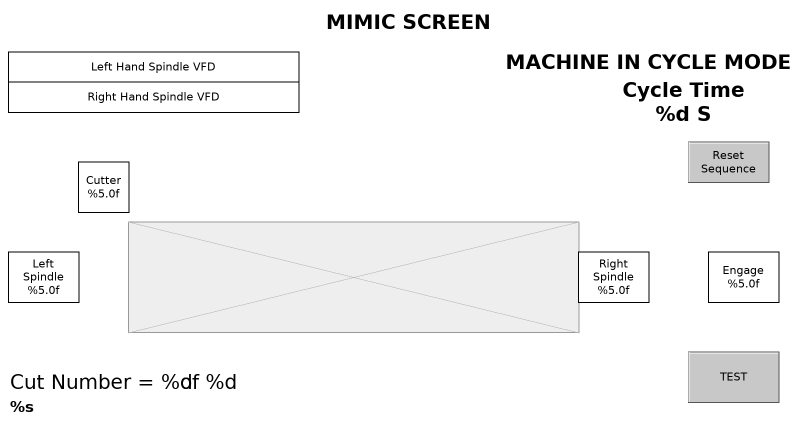
bitmap at (130,220)-(581,331): c:\users\graemep\pictures\bellow.bmp
rectangle at (80,160)-(131,211): text "Cutter / %5.0f"; shows MAIN.Axis[4].nActualPosition; x offset HMI.nCutterSlideXOffset; y offset HMI.nCutterYOffset; scale 1000
rectangle at (710,250)-(781,301): text "Engage / %5.0f"; shows MAIN.Axis[5].nActualPosition; x offset -HMI.nEnagageXOffset; y offset 0; scale 1000
rectangle at (580,250)-(651,301): text "Right / Spindle / %5.0f"; shows MAIN.Axis[2].nActualPosition; alarm colour if MAIN.bAxis2Coupled; x offset HMI.nRightSpindleXOffset; y offset 0; scale 1000
rectangle at (10,360)-(191,401): text "Cut Number = %d"; shows Sequencer.nCurrentCutNumber; invisible if .nMachineType = SIZER
button at (690,350)-(781,401): text "TEST"; invisible if .CurrentUserLevel < 2; taps Sequencer.bHMI_Overide
rectangle at (10,390)-(511,421): text "%s"; shows Sequencer.sSequence_Text
rounded rectangle at (10,50)-(301,81): text "Left Hand Spindle VFD"; invisible if .nMachineType = SIZER; alarm colour if .qbLeftHandSpindleOn
rounded rectangle at (10,80)-(301,111): text "Right Hand Spindle VFD"; invisible if .nMachineType = SIZER; alarm colour if .qbRightHandSpindleOn
rectangle at (10,250)-(81,301): text "Left / Spindle / %5.0f"; shows MAIN.Axis[1].nActualPosition; alarm colour if MAIN.bAxis2Coupled; x offset HMI.nLeftSpindleXOffset; y offset 0; scale 1000
rectangle at (500,40)-(801,81): text "MACHINE IN CYCLE MODE"; invisible if NOT MAIN.bInCycle
rectangle at (620,60)-(751,141): text "Cycle Time / %d S"; shows MAIN.nCycleTime
rectangle at (180,360)-(251,401): text "of %d"; shows .MachineRecipes[nCurrentRecipe].nNumberOfCuts; invisible if .nMachineType = SIZER
rectangle at (320,0)-(501,41): text "MIMIC SCREEN"
button at (690,140)-(771,181): text "Reset / Sequence"; runs INTERN ASSIGN Sequencer.nMachineSequence:=(0)
*)

(* Visualisation Helpers/Motion Helpers/MOVE_TABLE
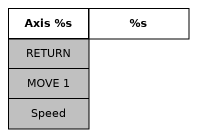
rounded rectangle at (0,30)-(81,61): text "RETURN"
rounded rectangle at (0,60)-(81,91): text "MOVE 1"
rounded rectangle at (0,0)-(81,31): text "Axis %s"; shows $AXISNUMBER$
rounded rectangle at (0,90)-(81,121): text "Speed"
rounded rectangle at (80,0)-(181,31): text "%s"; shows $AXISNAME$
3 elements of other kinds (tables, trends, ...) not read
*)

(* Visualisation Helpers/Motion Helpers/MUILTI_MOVE_TABLE
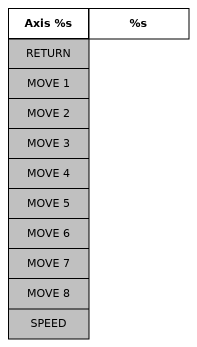
rounded rectangle at (0,30)-(81,61): text "RETURN"
rounded rectangle at (0,60)-(81,91): text "MOVE 1"
rounded rectangle at (0,90)-(81,121): text "MOVE 2"
rounded rectangle at (0,120)-(81,151): text "MOVE 3"
rounded rectangle at (0,150)-(81,181): text "MOVE 4"
rounded rectangle at (0,0)-(81,31): text "Axis %s"; shows $AXISNUMBER$
rounded rectangle at (0,300)-(81,331): text "SPEED"
rounded rectangle at (0,180)-(81,211): text "MOVE 5"
rounded rectangle at (0,210)-(81,241): text "MOVE 6"
rounded rectangle at (0,240)-(81,271): text "MOVE 7"
rounded rectangle at (0,270)-(81,301): text "MOVE 8"
rounded rectangle at (80,0)-(181,31): text "%s"; shows $AXISNAME$
10 elements of other kinds (tables, trends, ...) not read
*)

(* Visualisation Helpers/NUM_PAD
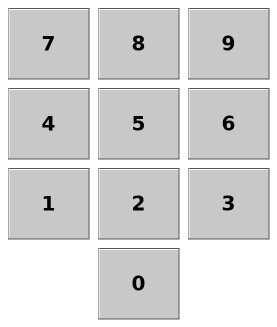
button at (20,20)-(101,91): text "7"; runs INTERN ASSIGN $KEY_PRESSED$:=(7)
button at (110,20)-(191,91): text "8"; runs INTERN ASSIGN $KEY_PRESSED$:=(8)
button at (110,260)-(191,331): text "0"; runs INTERN ASSIGN $KEY_PRESSED$:=(0)
button at (200,20)-(281,91): text "9"; runs INTERN ASSIGN $KEY_PRESSED$:=(9)
button at (20,100)-(101,171): text "4"; runs INTERN ASSIGN $KEY_PRESSED$:=(4)
button at (110,100)-(191,171): text "5"; runs INTERN ASSIGN $KEY_PRESSED$:=(5)
button at (200,100)-(281,171): text "6"; runs INTERN ASSIGN $KEY_PRESSED$:=(6)
button at (20,180)-(101,251): text "1"
button at (110,180)-(191,251): text "2"; runs INTERN ASSIGN $KEY_PRESSED$:=(2)
button at (200,180)-(281,251): text "3"; runs INTERN ASSIGN $KEY_PRESSED$:=(3)
*)

(* Visualisation Helpers/POPUP
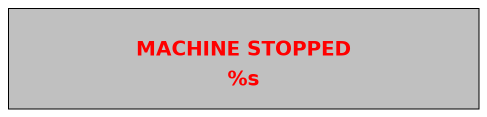
rectangle at (110,20)-(361,61): text "MACHINE STOPPED"; invisible if MAIN.bMachineRunning
rectangle at (20,50)-(451,91): text "%s"; shows Machine.ErrorHandler.sFirstError
2 more shapes without text or variables
*)

(* Visualisation RECIPE_EDITOR
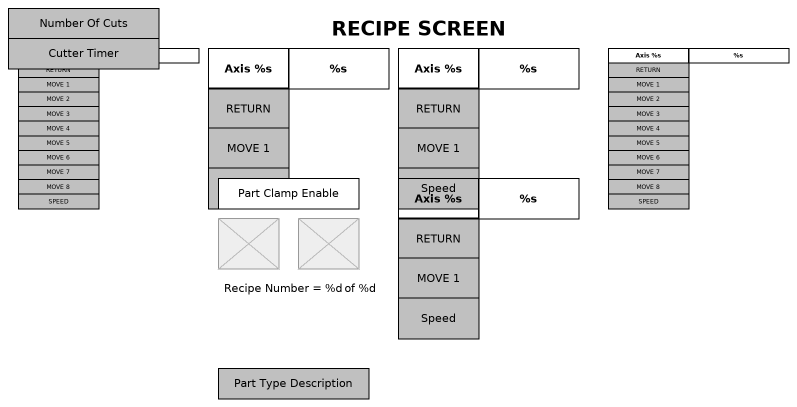
rectangle at (320,0)-(501,41): text "RECIPE SCREEN"
embedded screen at (10,40)-(191,201): MUILTI_MOVE_TABLE
embedded screen at (200,40)-(381,201): MOVE_TABLE
embedded screen at (390,40)-(571,201): MOVE_TABLE
bitmap at (210,210)-(271,261): c:\users\graemep\pictures\imagesi6yb17pr.jpg
bitmap at (290,210)-(351,261): c:\users\graemep\pictures\right arrow.jpg
rectangle at (200,260)-(351,301): text "Recipe Number = %d"; shows nRecipeNumber
embedded screen at (600,40)-(781,201): MUILTI_MOVE_TABLE
embedded screen at (390,170)-(571,331): MOVE_TABLE
rounded rectangle at (210,170)-(351,201): text "Part Clamp Enable"; invisible if .nMachineType = CUTTER; alarm colour if MachineRecipes[nRecipeNumber].bPartClampEnable; toggles MachineRecipes[nRecipeNumber].bPartClampEnable
rectangle at (330,260)-(371,301): text "of %d"; shows NUMBER_OF_RECIPES
rounded rectangle at (210,360)-(361,391): text "Part Type Description"
rounded rectangle at (0,0)-(151,31): text "Number Of Cycles"
rounded rectangle at (0,0)-(151,31): text "Number Of Cuts"
rounded rectangle at (0,30)-(151,61): text "Cutter Timer"
*)

(* Visualisation Helpers/Buttons/Round_Buttons/RED_IND_BTN_BMP_MOMENTRY
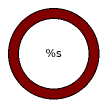
ellipse at (0,0)-(91,91): alarm colour if $INDICATOR$
ellipse at (10,10)-(81,81): text "%s"; shows $SWITCH_TITLE$; taps $SWITCH_INPUT$
*)

(* Visualisation Helpers/Buttons/Square_Buttons/RED_IND_SWITCH_BMP_MOMENTRY
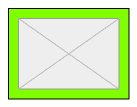
rounded rectangle at (0,0)-(121,91): alarm colour if $SWITCH_INPUT$
rounded rectangle at (10,10)-(111,81): taps $SWITCH_INPUT$
bitmap at (10,10)-(111,81): c:\users\graemep\pictures\right arrow.jpg
*)

(* Visualisation Helpers/Buttons/Square_Buttons/RED_IND_SWITCH_BMP_MTRY_LEFT
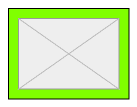
rounded rectangle at (0,0)-(121,91): alarm colour if $SWITCH_INPUT$
rounded rectangle at (10,10)-(111,81): taps $SWITCH_INPUT$
bitmap at (10,10)-(111,81): c:\users\graemep\pictures\imagesi6yb17pr.jpg
*)

(* Visualisation Helpers/Buttons/Square_Buttons/RED_INDICATOR_SWITCH_MOMENTRY
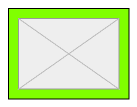
rounded rectangle at (0,0)-(121,91): alarm colour if $SWITCH_INPUT$
rounded rectangle at (10,10)-(111,81): text "%s"; shows $SWITCH_TITLE$; taps $SWITCH_INPUT$
bitmap at (10,10)-(111,81): $PICTURE$
*)

(* Visualisation Helpers/Buttons/Round_Buttons/RED_PUSH
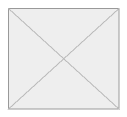
bitmap at (0,0)-(111,101): redup.bmp
bitmap at (0,0)-(111,101): reddown.bmp
*)

(* Visualisation SPLASH_SCREEN
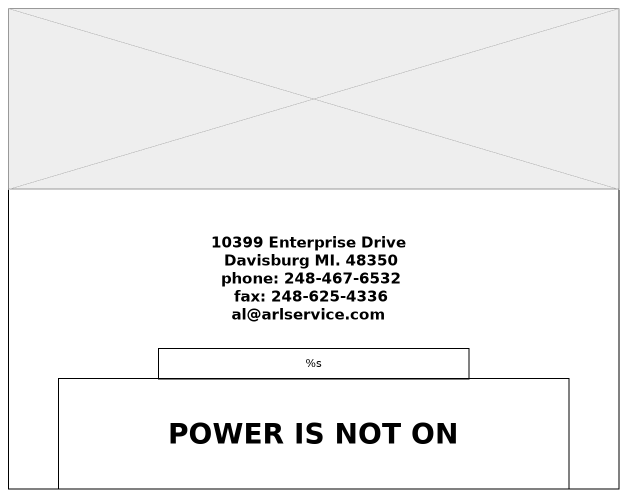
rectangle at (140,200)-(461,341): text "10399 Enterprise Drive / Davisburg MI. 48350 / phone: 248-467-6532 / fax: 248-625-4336 / al@arlservice.com"
bitmap at (0,0)-(611,181): c:\users\graemep\pictures\arl logo.bmp
rectangle at (50,370)-(561,481): text "POWER IS NOT ON"
rounded rectangle at (150,340)-(461,371): text "%s"; shows .VERSION_NUMBER
1 more shapes without text or variables
*)

(* Visualisation Helpers/Buttons/Square_Buttons/SWITCH_VISU
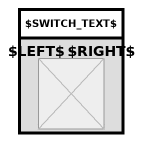
bitmap at (20,50)-(86,116): turnkeyon.bmp
rounded rectangle at (-5,25)-(41,61): text "$LEFT$"
rectangle at (0,0)-(106,31): text "$SWITCH_TEXT$"; alarm colour if $SWITCH_BOOL$
bitmap at (20,50)-(86,121): turnkeyoff.bmp
rounded rectangle at (60,25)-(106,61): text "$RIGHT$"
1 more shapes without text or variables
*)

(* Visualisation TC_VISU
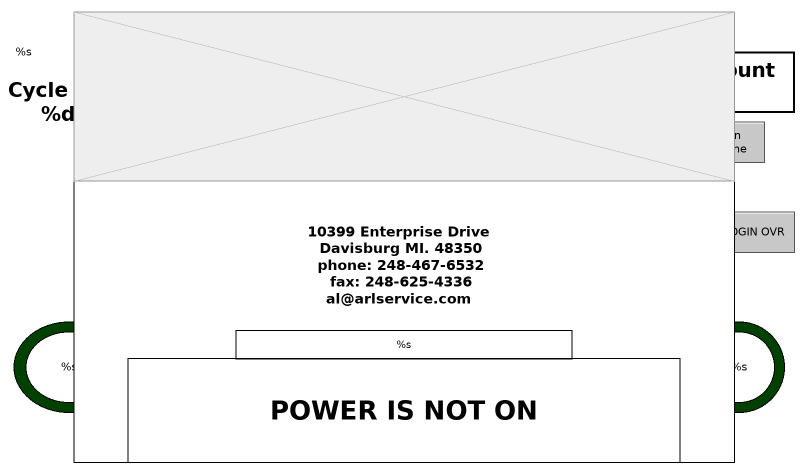
button at (710,210)-(791,251): text "LOGIN OVR"; runs INTERN ASSIGN CurrentUserLevel:=(4)
rectangle at (300,0)-(481,41): text "HOME SCREEN"
embedded screen at (210,320)-(321,431): YELOW_IND_BTN_BMP_MOMENTRY
embedded screen at (10,320)-(121,411): GREEN_IND_BTN_BMP_MOMENTRY
embedded screen at (110,320)-(221,421): RED_IND_BTN_BMP_MOMENTRY
embedded screen at (140,90)-(611,191): POPUP
rectangle at (250,110)-(501,151): text "MACHINE RUNNING"; invisible if NOT MAIN.bMachineRunning
embedded screen at (690,320)-(781,411): GREEN_IND_BTN_BMP_TOGGLE
rectangle at (240,200)-(541,241): text "MACHINE IN CYCLE MODE"; invisible if NOT MAIN.bInCycle
rounded rectangle at (620,50)-(791,111): text "Parts Count / %d"; shows nPartsCounter; runs INTERN ASSIGN nPartsCounter:=(0)
rectangle at (10,40)-(491,61): text "%s"; shows Sequencer.sSequence_Text
rounded rectangle at (210,240)-(361,271): text "Part Type Program"
rounded rectangle at (210,270)-(361,301): text "Part Type Description"
rectangle at (0,60)-(131,141): text "Cycle Time / %d S"; shows MAIN.nCycleTime
button at (680,120)-(761,161): text "Return / Machine"; taps Sequencer.bHMI_ReturnAll
embedded screen at (70,10)-(731,461): SPLASH_SCREEN
2 elements of other kinds (tables, trends, ...) not read
*)

(* Visualisation TEMPLATE
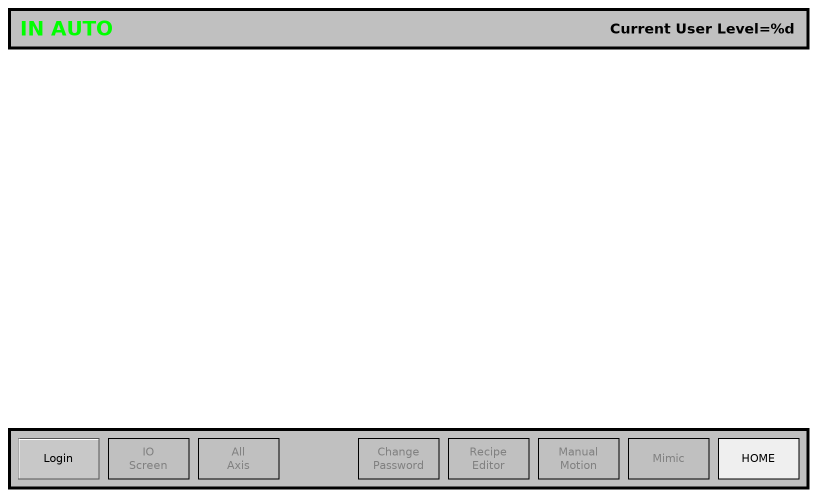
button at (440,430)-(521,471): text "Recipe / Editor"; opens RECIPE_EDITOR
button at (100,430)-(181,471): text "IO / Screen"; opens IO_SCREEN
button at (10,430)-(91,471): text "Login"; runs INTERN CHANGEUSERLEVEL
rectangle at (10,0)-(121,41): text "IN AUTO"; invisible if NOT .bAutomaticMode
button at (190,430)-(271,471): text "All / Axis"; opens ALL_AXIS
rectangle at (600,0)-(801,41): text "Current User Level=%d"; shows .CurrentUserLevel
button at (350,430)-(431,471): text "Change / Password"; invisible if .CurrentUserLevel < 2; runs INTERN CHANGEPASSWORD
button at (530,430)-(611,471): text "Manual / Motion"; opens MANUAL_MOTIONS
rectangle at (190,430)-(271,471): text "All / Axis"
rectangle at (440,430)-(521,471): text "Recipe / Editor"
rectangle at (350,430)-(431,471): text "Change / Password"
rectangle at (530,430)-(611,471): text "Manual / Motion"
rectangle at (100,430)-(181,471): text "IO / Screen"
button at (620,430)-(701,471): text "Mimic"; opens MIMIC
rectangle at (620,430)-(701,471): text "Mimic"
rectangle at (710,430)-(791,471): text "HOME"; invisible if HMI.bAtHomeScreen; alarm colour if Machine.ErrorHandler.bError_Present; opens TC_VISU
2 more shapes without text or variables
*)

(* Visualisation Helpers/Buttons/Round_Buttons/YEL_PUSH
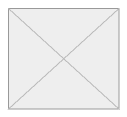
bitmap at (0,0)-(111,101): yellowup.bmp
bitmap at (0,0)-(111,101): yellowdown.bmp
*)

(* Visualisation Helpers/Buttons/Round_Buttons/YELOW_IND_BTN_BMP_MOMENTRY
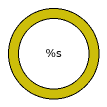
ellipse at (0,0)-(91,91): alarm colour if $INDICATOR$
ellipse at (10,10)-(81,81): taps $SWITCH_INPUT$
ellipse at (10,10)-(81,81): text "%s"; shows $SWITCH_TITLE$; taps $SWITCH_INPUT$
*)

(* Visualisation Helpers/Buttons/Round_Buttons/YELOW_IND_BTN_DL_MOMENTRY
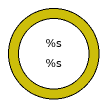
ellipse at (0,0)-(91,91): alarm colour if $INDICATOR$
ellipse at (10,10)-(81,81): taps $SWITCH_INPUT$
ellipse at (10,0)-(81,71): text "%s"; shows $SWITCH_TITLE1$; taps $SWITCH_INPUT$
ellipse at (10,20)-(81,91): text "%s"; shows $SWITCH_TITLE2$; taps $SWITCH_INPUT$
*)
